FUNCTION_BLOCK FB_AxisControl
VAR_INPUT
    bControlAllowed : BOOL;// 外部控制许可
	stLimit : ST_AxisLimit;// 当前轴的限位配置
    // 仅Clamping启用：使用驱动器6061确认真实CSP/CST状态。
    bUsePhysicalModeFeedback : BOOL;
    i8ModeOfOperationDisplay : SINT;
END_VAR

VAR_IN_OUT
    AxisRef : AXIS_REF;    // TwinCAT NC轴引用
    stAxis : ST_AxisInterface;    // 单轴命令、参数和反馈接口

END_VAR

VAR
    //==========================================================
    // PLCopen功能块实例
    //==========================================================

    fbPower   : MC_Power;
    fbReset   : MC_Reset;
    fbHome    : MC_Home;
    fbStop    : MC_Stop;
    fbJog     : MC_Jog;
    fbMoveAbs : MC_MoveAbsolute;
    fbMoveRel : MC_MoveRelative;
    fbTorqueControl : MC_TorqueControl;

    // 实际转矩达到阈值后的稳定确认。
    fbTorqueReached : TON;

    //==========================================================
    // 跨Method共享的内部运行状态
    //==========================================================

    stInternal : ST_AxisControlInternal;
	//==========================================================
    // 命令上升沿
    //
    // 所有R_TRIG必须在FB主体中每周期只调用一次。
    // 各执行方法只读取Q结果，不允许再次调用R_TRIG。
    //==========================================================

    trigReset   : R_TRIG;
    trigHome    : R_TRIG;
    trigMoveAbs : R_TRIG;
    trigMoveRel : R_TRIG;
    trigJogPos  : R_TRIG;
    trigJogNeg  : R_TRIG;


END_VAR

//==============================================================
// 0. 刷新NC轴状态
//
// AXIS_REF.Status不会自动周期刷新。
// 必须在读取Status.Error、Status.ErrorId和Status.Homed之前调用。
// 每根轴、每个PLC周期只能调用一次。
//==============================================================
M_ReadAxisStatus(
    ioAxisRef := AxisRef
);

//==============================================================
// 1. 清除上一个PLC周期的瞬时结果
//
// 必须在命令检测和执行方法之前调用。
// 后续方法可以在本周期重新设置完成、终止或拒绝信号。
//==============================================================

M_ClearCycleResults(
    ioAxis := stAxis
);


//==============================================================
// 2. 更新命令上升沿
//
// 必须在M_SelectCommand和所有执行方法之前调用。
//==============================================================

M_UpdateCommandEdges(
    iCmd := stAxis.ActiveCmd
);
//==============================================================
// 3. 更新软件限位状态
//
// 必须在点动和定位执行方法之前调用。
// 相对目标、绝对目标和点动方向许可均在此处计算。
//==============================================================

M_UpdateSoftLimitState(
    iLimit    := stLimit,
    ioAxisRef := AxisRef,
    ioAxis    := stAxis
);

//==============================================================
// 4. 汇总运动状态、生成停止请求并完成命令仲裁
//==============================================================
M_UpdateCommandArbitration(
    ioAxis := stAxis
);


//==============================================================
// 5. 调用四个执行方法
//
// 虽然命令已经完成仲裁，各MC功能块仍然必须每周期调用。
//==============================================================

// MC_Power必须每周期调用；同时处理Reset
M_ExecutePowerReset(
    ioAxisRef := AxisRef,
    ioAxis    := stAxis
);

// 执行MC_Home；只响应仲裁后的HomingCmd.bHome
M_ExecuteHoming(
    ioAxisRef := AxisRef,
    ioAxis    := stAxis
);

// 执行正向和负向点动
M_ExecuteJog(
    ioAxisRef := AxisRef,
    ioAxis    := stAxis
);

// 执行绝对运动和相对运动
M_ExecutePositioning(
    ioAxisRef := AxisRef,
    ioAxis    := stAxis
);

// 执行并保持转矩控制；撤销请求时由Stop恢复位置模式
M_ExecuteTorqueControl(
    ioAxisRef := AxisRef,
    ioAxis    := stAxis
);

// Stop最后调用，保证停止具有最终优先级
M_ExecuteStop(
    ioAxisRef := AxisRef,
    ioAxis    := stAxis
);

//==============================================================
// 6. 统一更新锁存错误
//
// 必须放在四个执行方法之后，以读取本周期最新的MC输出。
// 必须放在状态更新之前，因为bReady和eMotionState需要使用
// 最新的Alarm.bError。
//==============================================================

M_UpdateError(
    ioAxisRef := AxisRef,
    ioAxis    := stAxis
);


//==============================================================
// 7. 更新基础状态
//
// 必须在M_UpdateError之后调用，确保bReady使用本周期最新错误。
// 必须在运动状态更新之前调用，保证所有基础状态先完成刷新。
//==============================================================

M_UpdateBasicState(
    ioAxisRef := AxisRef,
    ioAxis    := stAxis
);


//==============================================================
// 8. 更新唯一运动状态
//
// 必须在M_UpdateError和M_UpdateBasicState之后调用。
//==============================================================

M_UpdateMotionState(
    ioAxisRef := AxisRef,
    ioAxis    := stAxis
);

//==============================================================
// 9. 更新轴实时数据
//
// 放在本周期调用链最后，向WPF提供最新的NC轴反馈。
//==============================================================

M_UpdateAxisData(
    ioAxisRef := AxisRef,
    ioAxis    := stAxis
);
//==============================================================
// 10. 更新运动方向
//
// 使用本周期最新的：
// 1. eMotionState；
// 2. fActVelocity；
// 3. fSetVelocity。
//
// 必须放在M_UpdateMotionState和M_UpdateAxisData之后。
//==============================================================

M_UpdateMotionDirection(
    ioAxis := stAxis
);

//==============================================================
// 方法名称：M_ClearCycleResults
// 功能：清除只保持一个PLC扫描周期的结果和提示信息
//
// 注意：
// 1. 本方法必须在每个PLC周期最开始调用；
// 2. 不清除bError、nErrorID和eErrorSource等锁存报警；
// 3. 锁存报警只能在MC_Reset成功后清除。
//==============================================================

METHOD PRIVATE M_ClearCycleResults

VAR_IN_OUT
    ioAxis : ST_AxisInterface;
    // 当前轴的命令、参数和反馈接口
END_VAR
//==============================================================
// 1. 清除单周期命令结果
//==============================================================

ioAxis.State.bDone := FALSE;
ioAxis.State.bCommandAborted := FALSE;
ioAxis.State.bCmdRejected := FALSE;


//==============================================================
// 2. 清除单周期拒绝原因
//==============================================================

ioAxis.Alarm.eRejectReason :=
    E_AxisRejectReason.NoReason;


//==============================================================
// 3. 清除单周期警告
//
// 当前警告没有采用锁存方式，因此每周期重新生成。
//==============================================================

ioAxis.Alarm.bWarning := FALSE;
ioAxis.Alarm.nWarningID := 0;
END_METHOD

//==============================================================
// 执行单轴回零命令
//
// DefaultHoming使用NC轴中已经完成的参考方式、方向、速度和
// 原点传感器映射。Direct只用于仿真建立临时参考坐标；
// ForceCalibration用于绝对编码器轴，不改变当前位置。
//==============================================================
METHOD PRIVATE M_ExecuteHoming
VAR_IN_OUT
    ioAxisRef : AXIS_REF;
    ioAxis    : ST_AxisInterface;
END_VAR
VAR
    eMcHomingMode : MC_HomingMode;
    bHomeAllowed  : BOOL;
END_VAR
CASE ioAxis.ActiveSet.Homing.eCommandMode OF
    E_AxisHomeCommandMode.Direct:
        eMcHomingMode := MC_Direct;

    E_AxisHomeCommandMode.ForceCalibration:
        eMcHomingMode := MC_ForceCalibration;

    ELSE
        eMcHomingMode := MC_DefaultHoming;
END_CASE;

bHomeAllowed :=
    bControlAllowed
    AND fbPower.Status
    AND NOT ioAxis.Alarm.bError
    AND NOT stInternal.bStopExecute
    AND NOT fbStop.Busy
    AND NOT fbReset.Busy
    AND NOT fbHome.Busy
    AND NOT stInternal.bHomeExecute
    AND NOT fbJog.Busy
    AND NOT fbMoveAbs.Busy
    AND NOT fbMoveRel.Busy
    AND NOT fbTorqueControl.Busy
    AND NOT fbTorqueControl.Active
    AND NOT stInternal.bMoveAbsExecute
    AND NOT stInternal.bMoveRelExecute
    AND NOT stInternal.bTorqueExecute;

IF trigHome.Q THEN
    IF bHomeAllowed
        AND (stInternal.eRequestedCommand = E_AxisCommand.Home)
    THEN
        stInternal.bHomeExecute := TRUE;
    ELSE
        ioAxis.State.bCmdRejected := TRUE;
        ioAxis.Alarm.eRejectReason :=
            E_AxisRejectReason.HomeNotAllowed;
    END_IF;
END_IF;

IF stInternal.bStopExecute THEN
    stInternal.bHomeExecute := FALSE;
END_IF;

fbHome(
    Axis       := ioAxisRef,
    Execute    := stInternal.bHomeExecute,
    Position   := ioAxis.ActiveSet.Homing.fReferencePosition,
    HomingMode := eMcHomingMode
);

IF fbHome.Done THEN
    stInternal.bHomeExecute := FALSE;
    ioAxis.State.bDone := TRUE;

ELSIF fbHome.CommandAborted THEN
    stInternal.bHomeExecute := FALSE;
    ioAxis.State.bCommandAborted := TRUE;

ELSIF fbHome.Error THEN
    stInternal.bHomeExecute := FALSE;
END_IF;
END_METHOD

//正反点动
METHOD PRIVATE M_ExecuteJog
VAR_IN_OUT
    ioAxisRef : AXIS_REF;
    // 当前Method使用的NC轴引用

    ioAxis : ST_AxisInterface;
    // 当前Method使用的单轴接口
END_VAR

VAR
    bJogAllowed       : BOOL;
    bJogDynamicsValid : BOOL;
    bJogForward       : BOOL;
    bJogBackward      : BOOL;
    bJogCommandEdge   : BOOL;
END_VAR
//==============================================================
// 1.根据仲裁结果生成MC_Jog方向
//
// 不再直接使用两个原始按钮驱动MC_Jog，
// 防止互斥命令或高优先级命令同时进入执行层。
//==============================================================

bJogForward :=
    stInternal.eRequestedCommand = E_AxisCommand.JogPositive;

bJogBackward :=
    stInternal.eRequestedCommand = E_AxisCommand.JogNegative;
bJogCommandEdge :=
    trigJogPos.Q
    OR trigJogNeg.Q;


//==============================================================
// 2. 检查点动参数
//==============================================================

bJogDynamicsValid :=
    ioAxis.ActiveSet.Jog.fVelocity > 0.0
    AND ioAxis.ActiveSet.Jog.fAcceleration >= 0.0
    AND ioAxis.ActiveSet.Jog.fDeceleration >= 0.0;

//==============================================================
// 4. 生成点动许可
//==============================================================

bJogAllowed :=
    bControlAllowed
    AND fbPower.Status
    AND NOT ioAxis.Alarm.bError
    AND NOT stInternal.bStopExecute
    AND NOT fbStop.Busy
    AND NOT fbReset.Busy
    AND NOT fbHome.Busy
    AND NOT stInternal.bHomeExecute
    AND NOT fbMoveAbs.Busy
    AND NOT fbMoveRel.Busy
    AND NOT stInternal.bMoveAbsExecute
    AND NOT stInternal.bMoveRelExecute
    AND bJogDynamicsValid;


//==============================================================
// 5. 点动命令拒绝
//
// 只在点动按钮产生上升沿时反馈一次拒绝结果。
// 点动运行过程中进入限位区时，MC_Jog方向输入会自动撤销。
//==============================================================

IF
    bJogCommandEdge
    AND ioAxis.ActiveCmd.bJogPos
    AND ioAxis.ActiveCmd.bJogNeg
THEN

    ioAxis.State.bCmdRejected := TRUE;

    ioAxis.Alarm.eRejectReason :=
        E_AxisRejectReason.JogDirectionConflict;


ELSIF
    bJogCommandEdge
    AND NOT bJogDynamicsValid
THEN

    ioAxis.State.bCmdRejected := TRUE;

    ioAxis.Alarm.eRejectReason :=
        E_AxisRejectReason.InvalidDynamics;


ELSIF
    bJogCommandEdge
    AND stInternal.stSoftLimitResult.bEnabled
    AND NOT stInternal.stSoftLimitResult.bConfigValid
THEN

    ioAxis.State.bCmdRejected := TRUE;

    ioAxis.Alarm.eRejectReason :=
        E_AxisRejectReason.SoftLimitConfigInvalid;


ELSIF
    bJogCommandEdge
    AND stInternal.stSoftLimitResult.bEnabled
    AND NOT stInternal.stSoftLimitResult.bReferenceValid
THEN

    ioAxis.State.bCmdRejected := TRUE;

    ioAxis.Alarm.eRejectReason :=
        E_AxisRejectReason.NotHomed;


ELSIF
    bJogCommandEdge
    AND
    (
        (
            ioAxis.ActiveCmd.bJogPos
            AND NOT stInternal.stSoftLimitResult.bJogPositiveAllowed
        )
        OR
        (
            ioAxis.ActiveCmd.bJogNeg
            AND NOT stInternal.stSoftLimitResult.bJogNegativeAllowed
        )
    )
THEN

    ioAxis.State.bCmdRejected := TRUE;

    ioAxis.Alarm.eRejectReason :=
        E_AxisRejectReason.TargetOutOfLimit;


ELSIF
    bJogCommandEdge
    AND NOT bJogAllowed
THEN

    ioAxis.State.bCmdRejected := TRUE;

    ioAxis.Alarm.eRejectReason :=
        E_AxisRejectReason.AxisNotReady;

END_IF;


//==============================================================
// 6. 周期调用MC_Jog
//==============================================================

fbJog(
    Axis := ioAxisRef,

    // 正向点动同时受到通用许可和正向软限位许可约束
    JogForward :=
        bJogAllowed
        AND bJogForward
        AND stInternal.stSoftLimitResult.bJogPositiveAllowed,

    // 负向点动同时受到通用许可和负向软限位许可约束
    JogBackwards :=
        bJogAllowed
        AND bJogBackward
        AND stInternal.stSoftLimitResult.bJogNegativeAllowed,

    Mode         := MC_JOGMODE_CONTINOUS,
    Position     := 0.0,
    Velocity     := ioAxis.ActiveSet.Jog.fVelocity,
    Acceleration := ioAxis.ActiveSet.Jog.fAcceleration,
    Deceleration := ioAxis.ActiveSet.Jog.fDeceleration,
    Jerk         := 0.0
);


//==============================================================
// 7. 点动被其他命令打断
//==============================================================

IF fbJog.CommandAborted THEN
    ioAxis.State.bCommandAborted := TRUE;
END_IF;
END_METHOD

//相对、绝对定位运动
METHOD PRIVATE M_ExecutePositioning
VAR_IN_OUT
    ioAxisRef : AXIS_REF;
    ioAxis    : ST_AxisInterface;
END_VAR

VAR
    bPositionAllowed       : BOOL;
    bPositionDynamicsValid : BOOL;
END_VAR
//==============================================================
// 1. 绝对/相对运动命令上升沿
//==============================================================



//==============================================================
// 2. 定位参数检查
//==============================================================

bPositionDynamicsValid :=
    ioAxis.ActiveSet.Position.fVelocity > 0.0
    AND ioAxis.ActiveSet.Position.fAcceleration >= 0.0
    AND ioAxis.ActiveSet.Position.fDeceleration >= 0.0;


//==============================================================
// 3. 统一定位许可
//==============================================================

bPositionAllowed :=
    bControlAllowed
    AND fbPower.Status
    AND ioAxis.State.bPositionModeReady
    AND NOT ioAxis.Alarm.bError
    AND NOT stInternal.bStopExecute
    AND NOT fbStop.Busy
    AND NOT fbReset.Busy
    AND NOT fbHome.Busy
    AND NOT stInternal.bHomeExecute
    AND NOT fbJog.Busy
    AND NOT ioAxis.ActiveCmd.bJogPos
    AND NOT ioAxis.ActiveCmd.bJogNeg
    AND NOT fbMoveAbs.Busy
    AND NOT fbMoveRel.Busy
    AND NOT stInternal.bMoveAbsExecute
    AND NOT stInternal.bMoveRelExecute;


//==============================================================
// 4. 接受或拒绝定位命令
//==============================================================

IF trigMoveAbs.Q AND trigMoveRel.Q THEN

    // 绝对和相对命令同时触发
    ioAxis.State.bCmdRejected := TRUE;

    ioAxis.Alarm.eRejectReason :=
        E_AxisRejectReason.CommandConflict;


ELSIF trigMoveAbs.Q OR trigMoveRel.Q THEN

    //==========================================================
    // 4.1 轴当前不允许定位
    //==========================================================

    IF NOT bPositionAllowed THEN

        ioAxis.State.bCmdRejected := TRUE;

        ioAxis.Alarm.eRejectReason :=
            E_AxisRejectReason.AxisNotReady;


    //==========================================================
    // 4.2 动态参数错误
    //==========================================================

    ELSIF NOT bPositionDynamicsValid THEN

        ioAxis.State.bCmdRejected := TRUE;

        ioAxis.Alarm.eRejectReason :=
            E_AxisRejectReason.InvalidDynamics;


    //==========================================================
    // 4.3 软件限位配置错误
    //==========================================================

    ELSIF
        stInternal.stSoftLimitResult.bEnabled
        AND NOT stInternal.stSoftLimitResult.bConfigValid
    THEN

        ioAxis.State.bCmdRejected := TRUE;

        ioAxis.Alarm.eRejectReason :=
            E_AxisRejectReason.SoftLimitConfigInvalid;


    //==========================================================
    // 4.4 尚未建立有效坐标基准
    //==========================================================

    ELSIF
        stInternal.stSoftLimitResult.bEnabled
        AND NOT stInternal.stSoftLimitResult.bReferenceValid
    THEN

        ioAxis.State.bCmdRejected := TRUE;

        ioAxis.Alarm.eRejectReason :=
            E_AxisRejectReason.NotHomed;


    //==========================================================
    // 4.5 绝对目标超出软件限位
    //==========================================================

    ELSIF
        stInternal.eRequestedCommand = E_AxisCommand.MoveAbsolute
        AND NOT stInternal.stSoftLimitResult.bAbsoluteTargetValid
    THEN

        ioAxis.State.bCmdRejected := TRUE;

        ioAxis.Alarm.eRejectReason :=
            E_AxisRejectReason.TargetOutOfLimit;


    //==========================================================
    // 4.6 相对运动最终目标超出软件限位
    //==========================================================

    ELSIF
        stInternal.eRequestedCommand = E_AxisCommand.MoveRelative
        AND NOT stInternal.stSoftLimitResult.bRelativeTargetValid
    THEN

        ioAxis.State.bCmdRejected := TRUE;

        ioAxis.Alarm.eRejectReason :=
            E_AxisRejectReason.TargetOutOfLimit;


    //==========================================================
    // 4.7 接受绝对运动
    //==========================================================

    ELSIF
        stInternal.eRequestedCommand = E_AxisCommand.MoveAbsolute
    THEN

        stInternal.bMoveAbsExecute := TRUE;


    //==========================================================
    // 4.8 接受相对运动
    //==========================================================

    ELSIF
        stInternal.eRequestedCommand = E_AxisCommand.MoveRelative
    THEN

        stInternal.bMoveRelExecute := TRUE;


    //==========================================================
    // 4.9 请求被高优先级命令覆盖
    //==========================================================

    ELSE

        ioAxis.State.bCmdRejected := TRUE;

        ioAxis.Alarm.eRejectReason :=
            E_AxisRejectReason.AxisNotReady;

    END_IF;

END_IF;


//==============================================================
// 5. Stop开始后撤销普通运动Execute
//==============================================================

IF stInternal.bStopExecute THEN
    stInternal.bHomeExecute := FALSE;
    stInternal.bMoveAbsExecute := FALSE;
    stInternal.bMoveRelExecute := FALSE;
    stInternal.bTorqueExecute := FALSE;
END_IF;


//==============================================================
// 6. 周期调用MC_MoveAbsolute
//==============================================================

fbMoveAbs(
    Axis         := ioAxisRef,
    Execute      := stInternal.bMoveAbsExecute,
    Position     := ioAxis.ActiveSet.Position.fAbsolutePosition,
    Velocity     := ioAxis.ActiveSet.Position.fVelocity,
    Acceleration := ioAxis.ActiveSet.Position.fAcceleration,
    Deceleration := ioAxis.ActiveSet.Position.fDeceleration,
    Jerk         := 0.0,
    BufferMode   := MC_Aborting
);


//==============================================================
// 7. 周期调用MC_MoveRelative
//==============================================================

fbMoveRel(
    Axis         := ioAxisRef,
    Execute      := stInternal.bMoveRelExecute,
    Distance     := ioAxis.ActiveSet.Position.fRelativeDistance,
    Velocity     := ioAxis.ActiveSet.Position.fVelocity,
    Acceleration := ioAxis.ActiveSet.Position.fAcceleration,
    Deceleration := ioAxis.ActiveSet.Position.fDeceleration,
    Jerk         := 0.0,
    BufferMode   := MC_Aborting
);


//==============================================================
// 8. 绝对运动结果
//==============================================================

IF fbMoveAbs.Done THEN

    stInternal.bMoveAbsExecute := FALSE;
    ioAxis.State.bDone := TRUE;

ELSIF fbMoveAbs.CommandAborted THEN

    stInternal.bMoveAbsExecute := FALSE;
    ioAxis.State.bCommandAborted := TRUE;

ELSIF fbMoveAbs.Error THEN

    stInternal.bMoveAbsExecute := FALSE;

END_IF;


//==============================================================
// 9. 相对运动结果
//==============================================================

IF fbMoveRel.Done THEN

    stInternal.bMoveRelExecute := FALSE;
    ioAxis.State.bDone := TRUE;

ELSIF fbMoveRel.CommandAborted THEN

    stInternal.bMoveRelExecute := FALSE;
    ioAxis.State.bCommandAborted := TRUE;

ELSIF fbMoveRel.Error THEN

    stInternal.bMoveRelExecute := FALSE;

END_IF;
END_METHOD

//==============================================================
// 执行持续型转矩控制。
// 撤销bTorqueControl后，命令仲裁会请求MC_Stop，
// 由NC将轴从CST恢复到位置相关模式。
//==============================================================
METHOD PRIVATE M_ExecuteTorqueControl
VAR_IN_OUT
    ioAxisRef : AXIS_REF;
    ioAxis    : ST_AxisInterface;
END_VAR

VAR
    bTorqueParametersValid : BOOL;
    bTorqueAllowed         : BOOL;
END_VAR
//==============================================================
// 1. 参数和执行许可
//==============================================================
bTorqueParametersValid :=
    ioAxis.ActiveSet.Torque.fMaxAbsTorquePercent > 0.0
    AND ABS(ioAxis.ActiveSet.Torque.fTargetTorquePercent)
        <= ioAxis.ActiveSet.Torque.fMaxAbsTorquePercent
    AND ioAxis.ActiveSet.Torque.fTorqueRampPercentPerSecond > 0.0
    AND ioAxis.ActiveSet.Torque.fVelocityLimitHigh > 0.0
    AND ioAxis.ActiveSet.Torque.fVelocityLimitLow < 0.0
    AND ioAxis.ActiveSet.Torque.fVelocityLimitHigh
        > ioAxis.ActiveSet.Torque.fVelocityLimitLow;

bTorqueAllowed :=
    bControlAllowed
    AND fbPower.Status
    AND NOT ioAxis.Alarm.bError
    AND NOT stInternal.bStopExecute
    AND NOT fbStop.Busy
    AND NOT fbReset.Busy
    AND NOT fbHome.Busy
    AND NOT stInternal.bHomeExecute
    AND NOT fbJog.Busy
    AND NOT fbMoveAbs.Busy
    AND NOT fbMoveRel.Busy
    AND NOT stInternal.bMoveAbsExecute
    AND NOT stInternal.bMoveRelExecute;

//==============================================================
// 2. 接受、保持或撤销转矩命令
//==============================================================
IF
    NOT ioAxis.ActiveCmd.bTorqueControl
    OR
    (stInternal.eRequestedCommand <> E_AxisCommand.TorqueControl)
THEN
    stInternal.bTorqueExecute := FALSE;

ELSIF NOT stInternal.bTorqueExecute THEN
    IF NOT bTorqueAllowed THEN
        ioAxis.State.bCmdRejected := TRUE;
        ioAxis.Alarm.eRejectReason :=
            E_AxisRejectReason.AxisNotReady;

    ELSIF NOT bTorqueParametersValid THEN
        ioAxis.State.bCmdRejected := TRUE;
        ioAxis.Alarm.eRejectReason :=
            E_AxisRejectReason.InvalidDynamics;

    ELSE
        stInternal.bTorqueExecute := TRUE;
    END_IF;
END_IF;

//==============================================================
// 3. 周期调用MC_TorqueControl
//==============================================================
fbTorqueControl(
    Axis              := ioAxisRef,
    Execute           := stInternal.bTorqueExecute,
    ContinuousUpdate  := TRUE,
    Relative          := FALSE,
    Torque            := ioAxis.ActiveSet.Torque.fTargetTorquePercent,
    TorqueRamp        := ioAxis.ActiveSet.Torque.fTorqueRampPercentPerSecond,
    VelocityLimitHigh := ioAxis.ActiveSet.Torque.fVelocityLimitHigh,
    VelocityLimitLow  := ioAxis.ActiveSet.Torque.fVelocityLimitLow,
    BufferMode        := MC_Aborting
);

//==============================================================
// 4. 实际转矩稳定确认
//==============================================================
fbTorqueReached(
    IN :=
        fbTorqueControl.Active
        AND
        (
            ABS(ioAxis.Data.fActTorque)
            >= ioAxis.ActiveSet.Torque.fReachedMinAbsTorquePercent
        ),
    PT := ioAxis.ActiveSet.Torque.tReachedStableTime
);

ioAxis.State.bTorqueReached := fbTorqueReached.Q;
ioAxis.State.bTorqueControlActive := fbTorqueControl.Active;

//==============================================================
// 5. 发布当前控制模式
//==============================================================
IF bUsePhysicalModeFeedback THEN
    // Clamping必须以驱动器6061为准，不能由PLCopen FB内部状态推断。
    CASE i8ModeOfOperationDisplay OF
        8:
            ioAxis.State.eControlMode := E_AxisControlMode.Position;
        10:
            ioAxis.State.eControlMode := E_AxisControlMode.Torque;
        ELSE
            ioAxis.State.eControlMode := E_AxisControlMode.Undefined;
    END_CASE;
ELSE
    IF fbTorqueControl.Active OR fbTorqueControl.Busy THEN
        ioAxis.State.eControlMode := E_AxisControlMode.Torque;
    ELSIF
        fbPower.Status
        AND NOT stInternal.bStopExecute
        AND NOT fbStop.Busy
    THEN
        ioAxis.State.eControlMode := E_AxisControlMode.Position;
    ELSE
        ioAxis.State.eControlMode := E_AxisControlMode.Undefined;
    END_IF;
END_IF;

ioAxis.State.bPositionModeReady :=
    fbPower.Status
    AND (ioAxis.State.eControlMode = E_AxisControlMode.Position)
    AND NOT stInternal.bStopExecute
    AND NOT fbStop.Busy;

ioAxis.State.bTorqueModeReady :=
    fbTorqueControl.Active
    AND (ioAxis.State.eControlMode = E_AxisControlMode.Torque);

//==============================================================
// 6. 功能块结果
//==============================================================
IF fbTorqueControl.CommandAborted THEN
    stInternal.bTorqueExecute := FALSE;
    ioAxis.State.bCommandAborted := TRUE;
ELSIF fbTorqueControl.Error THEN
    stInternal.bTorqueExecute := FALSE;
END_IF;
END_METHOD

//调用 MC_Power和MC_Reset
METHOD PRIVATE M_ExecutePowerReset
VAR_IN_OUT
    ioAxisRef : AXIS_REF;
    ioAxis    : ST_AxisInterface;
END_VAR

VAR
    bPowerEnable  : BOOL; // 实际送入MC_Power的Enable
    bResetAllowed : BOOL; // 当前是否允许复位	
END_VAR
//==============================================================
// 1. 生成MC_Power实际使能信号
//
// 外部要求使能时正常保持使能。
// 运动中撤销使能时，先保持使能完成MC_Stop。
//==============================================================

bPowerEnable :=
    ioAxis.ActiveCmd.bEnable
    OR
    (
        (stInternal.bStopExecute OR fbStop.Busy)
        AND fbPower.Status
    );


//==============================================================
// 2. 周期调用MC_Power
//==============================================================

fbPower(
    Axis            := ioAxisRef,
    Enable          := bPowerEnable,
    Enable_Positive := TRUE,
    Enable_Negative := TRUE,
    Override        := 100.0
);



//==============================================================
// 3. Reset许可
//
// 运动、点动和停止过程中不允许Reset。
//==============================================================

bResetAllowed :=
    NOT stInternal.bMotionActive
    AND NOT stInternal.bStopExecute
    AND NOT fbStop.Busy;

//==============================================================
// 4. 周期调用MC_Reset
//
// Reset必须同时满足：
// 1. 已被M_SelectCommand选中；
// 2. 当前轴状态允许复位。
//==============================================================

fbReset(
    Axis := ioAxisRef,
    Execute :=
        (stInternal.eRequestedCommand = E_AxisCommand.Reset)
        AND bResetAllowed
);


//==============================================================
// 5. Reset命令被拒绝
//==============================================================

IF
    (stInternal.eRequestedCommand = E_AxisCommand.Reset)
    AND NOT bResetAllowed
THEN
    ioAxis.State.bCmdRejected := TRUE;

    ioAxis.Alarm.eRejectReason :=
        E_AxisRejectReason.ResetDuringMotion;
END_IF;

//==============================================================
// 6. Reset成功
//
// 清除PLC锁存的轴报警。
//==============================================================

IF fbReset.Done THEN

    ioAxis.Alarm.bError       := FALSE;
    ioAxis.Alarm.nErrorID     := 0;
    ioAxis.Alarm.eErrorSource :=
        E_AxisErrorSource.NoError;

    ioAxis.State.bDone := TRUE;

END_IF;
END_METHOD

//处理最高优先级停止和 MC_Stop
METHOD PRIVATE M_ExecuteStop
VAR_IN_OUT
    ioAxisRef : AXIS_REF;
    ioAxis    : ST_AxisInterface;
END_VAR

VAR
    fStopDeceleration : LREAL;//停止声明
END_VAR
//==============================================================
// 1. Stop开始后撤销定位和转矩Execute
//==============================================================
IF stInternal.bStopExecute THEN
    stInternal.bHomeExecute := FALSE;
    stInternal.bMoveAbsExecute := FALSE;
    stInternal.bMoveRelExecute := FALSE;
    stInternal.bTorqueExecute := FALSE;
END_IF;


//==============================================================
// 2. 选择停止减速度
//
// 当前沿用位置运动减速度。
// 如果配置值小于0，则使用0，让NC采用默认减速度。
//==============================================================
fStopDeceleration :=
    ioAxis.ActiveSet.Position.fDeceleration;

IF fStopDeceleration < 0.0 THEN
    fStopDeceleration := 0.0;
END_IF;


//==============================================================
// 3. 每周期调用MC_Stop
//==============================================================
fbStop(
    Axis         := ioAxisRef,
    Execute      := stInternal.bStopExecute,
    Deceleration := fStopDeceleration,
    Jerk         := 0.0
);


//==============================================================
// 4. 发布MC_Stop专用状态
//
// 不使用通用State.bDone，避免与MoveAbs、MoveRel等完成信号混淆。
//==============================================================
ioAxis.State.bStopDone :=
    fbStop.Done;

// Done仅代表停住；释放Execute并等待Busy结束后才能掉使能。
ioAxis.State.bStopReleased :=
    NOT stInternal.bStopExecute
    AND NOT fbStop.Busy;

ioAxis.State.bStopError :=
    fbStop.Error;

ioAxis.State.nStopErrorID :=
    fbStop.ErrorID;


//==============================================================
// 5. 外部停止请求释放后，解除MC_Stop锁定
//==============================================================
IF
    fbStop.Done
    AND NOT stInternal.bStopRequest
THEN
    stInternal.bStopExecute := FALSE;
END_IF;


//==============================================================
// 6. Stop错误
//
// 即使停止发生错误，也要撤销内部Execute，
// 错误信息由State和Alarm继续对外发布。
//==============================================================
IF fbStop.Error THEN
    stInternal.bStopExecute := FALSE;
END_IF;
END_METHOD

// 刷新NC轴状态。每根轴、每周期只调用一次。
METHOD PRIVATE M_ReadAxisStatus
VAR_IN_OUT
    ioAxisRef : AXIS_REF;
END_VAR
ioAxisRef.ReadStatus();
END_METHOD

//==============================================================
// 方法名称：M_SelectCommand
// 功能：
// 1. 识别外部BOOL命令；
// 2. 将多个BOOL命令转换成唯一E_AxisCommand；
// 3. 实现停止、复位、点动、定位之间的优先级；
// 4. 发现互斥命令时返回NoCommand。
//
// 本方法只进行命令选择，不调用任何MC功能块。
//==============================================================

METHOD PRIVATE M_SelectCommand : E_AxisCommand

VAR_INPUT
    bStopRequest  : BOOL; // 停止请求，最高优先级
    bResetPulse   : BOOL; // 复位命令上升沿

    bHomePulse    : BOOL; // 回零命令上升沿

    bTorqueControl : BOOL; // 持续型转矩控制请求

    bJogPositive  : BOOL; // 正向点动保持信号
    bJogNegative  : BOOL; // 负向点动保持信号

    bMoveAbsPulse : BOOL; // 绝对运动命令上升沿
    bMoveRelPulse : BOOL; // 相对运动命令上升沿
END_VAR
// 默认本周期没有有效命令
M_SelectCommand := E_AxisCommand.NoCommand;


//==============================================================
// 1. 停止命令
//
// Stop具有最高优先级，可以覆盖复位、点动和定位命令。
// bStopRequest还包括撤销控制许可和运动中撤销使能。
//==============================================================

IF bStopRequest THEN

    M_SelectCommand := E_AxisCommand.Stop;


//==============================================================
// 2. 复位命令
//
// Reset使用上升沿，只在触发周期返回Reset。
// 是否允许复位仍由M_ExecutePowerReset检查。
//==============================================================

ELSIF bResetPulse THEN

    M_SelectCommand := E_AxisCommand.Reset;


//==============================================================
// 3. 回零命令
//==============================================================

ELSIF bHomePulse THEN

    M_SelectCommand := E_AxisCommand.Home;


//==============================================================
// 4. 转矩控制
//==============================================================

ELSIF bTorqueControl THEN

    M_SelectCommand := E_AxisCommand.TorqueControl;


//==============================================================
// 4. 点动方向冲突
//
// 正向点动和负向点动同时成立时不选择任何方向。
// 具体拒绝原因由M_ExecuteJog写入状态和报警接口。
//==============================================================

ELSIF bJogPositive AND bJogNegative THEN

    M_SelectCommand := E_AxisCommand.NoCommand;


//==============================================================
// 5. 正向和负向点动
//
// 点动是保持型命令：
// 按钮保持TRUE时，每周期持续返回对应点动命令；
// 松开按钮后返回NoCommand，MC_Jog开始减速停止。
//==============================================================

ELSIF bJogPositive THEN

    M_SelectCommand := E_AxisCommand.JogPositive;

ELSIF bJogNegative THEN

    M_SelectCommand := E_AxisCommand.JogNegative;


//==============================================================
// 6. 定位命令冲突
//
// 绝对运动和相对运动在同一扫描周期同时触发时，
// 不选择任何定位命令。
// 具体拒绝原因由M_ExecutePositioning写入反馈。
//==============================================================

ELSIF bMoveAbsPulse AND bMoveRelPulse THEN

    M_SelectCommand := E_AxisCommand.NoCommand;


//==============================================================
// 7. 绝对运动和相对运动
//==============================================================

ELSIF bMoveAbsPulse THEN

    M_SelectCommand := E_AxisCommand.MoveAbsolute;

ELSIF bMoveRelPulse THEN

    M_SelectCommand := E_AxisCommand.MoveRelative;

END_IF;
END_METHOD

//==============================================================
// 方法名称：M_UpdateAxisData
// 功能：
// 1. 从AXIS_REF.NcToPlc读取NC轴实时数据；
// 2. 写入ST_AxisData，供PLC程序和WPF读取；
// 3. 集中处理后续可能增加的单位换算。
//
// 调用位置：
// 放在所有命令执行、错误和状态更新之后，每周期调用一次。
//==============================================================

METHOD PRIVATE M_UpdateAxisData

VAR_IN_OUT
    ioAxisRef : AXIS_REF;
    // 当前TwinCAT NC轴引用

    ioAxis : ST_AxisInterface;
    // 当前单轴数据反馈接口
END_VAR
//==============================================================
// 1. 位置数据
//==============================================================

// NC轴设定位置
ioAxis.Data.fSetPosition :=
    ioAxisRef.NcToPlc.SetPos;

// 编码器反馈的实际位置
ioAxis.Data.fActPosition :=
    ioAxisRef.NcToPlc.ActPos;

// 当前运动的目标位置
ioAxis.Data.fTargetPosition :=
    ioAxisRef.NcToPlc.TargetPos;


//==============================================================
// 2. 速度数据
//==============================================================

// NC轴设定速度
ioAxis.Data.fSetVelocity :=
    ioAxisRef.NcToPlc.SetVelo;

// 编码器反馈的实际速度
ioAxis.Data.fActVelocity :=
    ioAxisRef.NcToPlc.ActVelo;


//==============================================================
// 3. 加速度数据
//==============================================================

// NC轴设定加速度
ioAxis.Data.fSetAcceleration :=
    ioAxisRef.NcToPlc.SetAcc;

// NC轴实际加速度
ioAxis.Data.fActAcceleration :=
    ioAxisRef.NcToPlc.ActAcc;


//==============================================================
// 4. 跟随误差
//
// 带方向的位置偏差。
//==============================================================

ioAxis.Data.fFollowingError :=
    ioAxisRef.NcToPlc.PosDiff;


//==============================================================
// 5. 转矩数据
//
// 是否为实际物理转矩、百分比或归一化值，
// 取决于驱动器和NC轴的配置。
//==============================================================

ioAxis.Data.fSetTorque :=
    ioAxisRef.NcToPlc.SetTorque;

ioAxis.Data.fActTorque :=
    ioAxisRef.NcToPlc.ActTorque;


//==============================================================
// 6. 电机转速
//
// 当前缺少“每转对应多少工程单位”的换算参数，
// 因此暂不计算实际rpm。
//==============================================================

ioAxis.Data.fActRpm := 0.0;
END_METHOD

//==============================================================
// 方法名称：M_UpdateBasicState
// 功能：
// 1. 汇总各PLCopen功能块的Busy状态；
// 2. 更新轴使能、忙碌、活动、准备完成和回零状态；
// 3. 为WPF提供统一的基础状态反馈。
//
// 调用位置：
// 必须放在四个执行方法和M_UpdateError之后。
//==============================================================

METHOD PRIVATE M_UpdateBasicState

VAR_IN_OUT
    ioAxisRef : AXIS_REF;
    // 当前TwinCAT NC轴引用

    ioAxis : ST_AxisInterface;
    // 当前单轴状态和报警接口
END_VAR
//==============================================================
// 1. 汇总轴忙碌状态
//
// 除PLCopen功能块的Busy外，还包含三个Execute锁存信号，
// 避免命令已经接受但Busy尚未建立时出现一周期状态空缺。
//==============================================================

stInternal.bAnyBusy :=
    fbReset.Busy
    OR fbHome.Busy
    OR stInternal.bHomeExecute
    OR fbStop.Busy
    OR stInternal.bStopExecute
    OR fbJog.Busy
    OR fbMoveAbs.Busy
    OR fbMoveRel.Busy
    OR fbTorqueControl.Busy
    OR stInternal.bMoveAbsExecute
    OR stInternal.bMoveRelExecute
    OR stInternal.bTorqueExecute;


//==============================================================
// 2. 更新实际使能状态
//
// 采用MC_Power.Status，而不是外部bEnable请求。
//==============================================================

ioAxis.State.bPowerStatus :=
    fbPower.Status;


//==============================================================
// 3. 更新忙碌状态
//
// 复位、停止、点动或定位过程中均视为Busy。
//==============================================================

ioAxis.State.bBusy :=
    stInternal.bAnyBusy;


//==============================================================
// 4. 更新有效运动状态
//
// bActive表示NC轴当前存在实际运动或停止过程。
// 不包含仅已锁存、但PLCopen Busy尚未建立的命令。
//==============================================================

ioAxis.State.bActive :=
    fbJog.Busy
    OR fbHome.Busy
    OR fbMoveAbs.Busy
    OR fbMoveRel.Busy
    OR fbTorqueControl.Active
    OR fbStop.Busy;


//==============================================================
// 5. 更新轴准备状态
//
// 满足以下全部条件才允许接受新的普通运动命令：
// 1. 轴已经实际使能；
// 2. 外部控制许可有效；
// 3. 没有锁存错误；
// 4. 当前没有正在执行的命令。
//==============================================================

ioAxis.State.bReady :=
    fbPower.Status
    AND bControlAllowed
    AND NOT ioAxis.Alarm.bError
    AND NOT stInternal.bAnyBusy;


//==============================================================
// 6. 更新回零状态
//
// MC_Home和NC轴状态共同维护该标志。
//==============================================================

ioAxis.State.bHomed :=
    ioAxisRef.Status.Homed;
END_METHOD

//==============================================================
// 汇总运动状态、生成停止请求、选择唯一命令并锁存停止。
//==============================================================
METHOD PRIVATE M_UpdateCommandArbitration
VAR_IN_OUT
    ioAxis : ST_AxisInterface;
END_VAR
// Execute已锁存但Busy尚未建立时，同样视为运动有效。
stInternal.bMotionActive :=
    fbJog.Busy
    OR fbHome.Busy
    OR fbMoveAbs.Busy
    OR fbMoveRel.Busy
    OR fbTorqueControl.Active
    OR fbTorqueControl.Busy
    OR stInternal.bMoveAbsExecute
    OR stInternal.bMoveRelExecute
    OR stInternal.bHomeExecute
    OR stInternal.bTorqueExecute;


// 外部Stop、运动中撤销控制许可或撤销使能均请求停止。
stInternal.bStopRequest :=
    ioAxis.ActiveCmd.bStop
    OR
    (
        (fbTorqueControl.Active OR fbTorqueControl.Busy)
        AND NOT ioAxis.ActiveCmd.bTorqueControl
    )
    OR
    (
        NOT bControlAllowed
        AND stInternal.bMotionActive
    )
    OR
    (
        NOT ioAxis.ActiveCmd.bEnable
        AND stInternal.bMotionActive
    );


// 优先级：Stop > Reset > Torque > Jog > MoveAbsolute/MoveRelative。
stInternal.eRequestedCommand := M_SelectCommand(
    bStopRequest := stInternal.bStopRequest,
    bResetPulse := trigReset.Q,
    bHomePulse := trigHome.Q,
    bTorqueControl := ioAxis.ActiveCmd.bTorqueControl,
    bJogPositive := ioAxis.ActiveCmd.bJogPos,
    bJogNegative := ioAxis.ActiveCmd.bJogNeg,
    bMoveAbsPulse := trigMoveAbs.Q,
    bMoveRelPulse := trigMoveRel.Q
);


// Stop一旦被选中，保持Execute直至停止完成并释放外部Stop。
IF
    (stInternal.eRequestedCommand = E_AxisCommand.Stop)
    AND fbPower.Status
THEN
    stInternal.bStopExecute := TRUE;
END_IF;
END_METHOD

//==============================================================
// 方法名称：M_UpdateCommandEdges
// 功能：统一更新单轴命令的上升沿检测结果
//
// 注意：
// 1. 每个R_TRIG实例每周期只能在本方法中调用一次；
// 2. Reset、绝对运动、相对运动使用上升沿触发；
// 3. 点动使用持续信号，上升沿仅用于判断命令是否被拒绝；
// 4. Enable和Stop是持续型信号，不需要R_TRIG。
//==============================================================

METHOD PRIVATE M_UpdateCommandEdges

VAR_INPUT
    iCmd : ST_AxisCmd;
    // 当前轴的原始命令
    // 结构体较小，使用VAR_INPUT传递不会造成明显开销
END_VAR
//==============================================================
// 1. 错误复位命令上升沿
//==============================================================

trigReset(
    CLK := iCmd.bReset
);


//==============================================================
// 2. 回零命令上升沿
//==============================================================

trigHome(
    CLK := iCmd.bHome
);


//==============================================================
// 3. 绝对运动命令上升沿
//==============================================================

trigMoveAbs(
    CLK := iCmd.bMoveAbs
);


//==============================================================
// 3. 相对运动命令上升沿
//==============================================================

trigMoveRel(
    CLK := iCmd.bMoveRel
);


//==============================================================
// 4. 正向点动按钮上升沿
//
// MC_Jog仍然使用bJogPos持续电平；
// 本上升沿只用于产生命令拒绝反馈。
//==============================================================

trigJogPos(
    CLK := iCmd.bJogPos
);


//==============================================================
// 5. 负向点动按钮上升沿
//==============================================================

trigJogNeg(
    CLK := iCmd.bJogNeg
);
END_METHOD

//==============================================================
// 方法名称：M_UpdateError
// 功能：
// 1. 汇总NC轴和各PLCopen功能块错误；
// 2. 根据优先级选择当前显示的错误；
// 3. 将错误锁存到单轴报警接口。
//
// 错误优先级：
// NC轴 > Stop > Power > Reset > Jog > 绝对运动 > 相对运动
//
// 注意：
// 1. 本方法不主动清除错误；
// 2. 错误只能在MC_Reset成功后清除；
// 3. 没有新错误时保持原报警不变。
//==============================================================

METHOD PRIVATE M_UpdateError

VAR_IN_OUT
    ioAxisRef : AXIS_REF;
    // 当前TwinCAT NC轴引用

    ioAxis : ST_AxisInterface;
    // 当前轴的状态和报警接口
END_VAR
//==============================================================
// 1. NC轴错误
//
// NC轴本体错误优先级最高。
//==============================================================

IF ioAxisRef.Status.Error THEN

    ioAxis.Alarm.bError := TRUE;
    ioAxis.Alarm.nErrorID :=
        ioAxisRef.Status.ErrorId;

    ioAxis.Alarm.eErrorSource :=
        E_AxisErrorSource.NcAxis;


//==============================================================
// 2. MC_Stop错误
//==============================================================

ELSIF fbStop.Error THEN

    ioAxis.Alarm.bError := TRUE;
    ioAxis.Alarm.nErrorID :=
        fbStop.ErrorID;

    ioAxis.Alarm.eErrorSource :=
        E_AxisErrorSource.Stop;


//==============================================================
// 3. MC_Power错误
//==============================================================

ELSIF fbPower.Error THEN

    ioAxis.Alarm.bError := TRUE;
    ioAxis.Alarm.nErrorID :=
        fbPower.ErrorID;

    ioAxis.Alarm.eErrorSource :=
        E_AxisErrorSource.Power;


//==============================================================
// 4. MC_Reset错误
//==============================================================

ELSIF fbReset.Error THEN

    ioAxis.Alarm.bError := TRUE;
    ioAxis.Alarm.nErrorID :=
        fbReset.ErrorID;

    ioAxis.Alarm.eErrorSource :=
        E_AxisErrorSource.Reset;


//==============================================================
// 5. MC_Home错误
//==============================================================

ELSIF fbHome.Error THEN

    ioAxis.Alarm.bError := TRUE;
    ioAxis.Alarm.nErrorID :=
        fbHome.ErrorID;

    ioAxis.Alarm.eErrorSource :=
        E_AxisErrorSource.Home;


//==============================================================
// 6. MC_TorqueControl错误
//==============================================================

ELSIF fbTorqueControl.Error THEN

    ioAxis.Alarm.bError := TRUE;
    ioAxis.Alarm.nErrorID :=
        fbTorqueControl.ErrorID;

    ioAxis.Alarm.eErrorSource :=
        E_AxisErrorSource.TorqueControl;


//==============================================================
// 6. MC_Jog错误
//==============================================================

ELSIF fbJog.Error THEN

    ioAxis.Alarm.bError := TRUE;
    ioAxis.Alarm.nErrorID :=
        fbJog.ErrorID;

    ioAxis.Alarm.eErrorSource :=
        E_AxisErrorSource.Jog;


//==============================================================
// 7. MC_MoveAbsolute错误
//==============================================================

ELSIF fbMoveAbs.Error THEN

    ioAxis.Alarm.bError := TRUE;
    ioAxis.Alarm.nErrorID :=
        fbMoveAbs.ErrorID;

    ioAxis.Alarm.eErrorSource :=
        E_AxisErrorSource.MoveAbsolute;


//==============================================================
// 8. MC_MoveRelative错误
//==============================================================

ELSIF fbMoveRel.Error THEN

    ioAxis.Alarm.bError := TRUE;
    ioAxis.Alarm.nErrorID :=
        fbMoveRel.ErrorID;

    ioAxis.Alarm.eErrorSource :=
        E_AxisErrorSource.MoveRelative;

END_IF;
END_METHOD

//==============================================================
// 方法名称：M_UpdateMotionDirection
//
// 功能：
// 1. 根据轴当前运动状态判断是否需要输出运动方向；
// 2. 优先使用NC实际速度判断方向；
// 3. 运动刚启动、实际速度尚未建立时，使用NC设定速度辅助判断；
// 4. 停止、故障、未使能等状态统一输出None；
// 5. 不使用目标位置，避免中途停止后旧目标造成方向状态残留。
//
// 调用位置：
// 必须在M_UpdateMotionState和M_UpdateAxisData之后调用。
//==============================================================

METHOD PRIVATE M_UpdateMotionDirection

VAR_IN_OUT
    ioAxis : ST_AxisInterface;
    // 当前单轴命令、数据和状态接口
END_VAR

VAR CONSTANT
    // 速度方向判断死区。
    //
    // 防止轴在零速附近因浮点波动频繁切换正负方向。
    // 当前单位取决于具体业务轴的工程单位，直线轴通常为mm/s。
    c_fVelocityDeadband : LREAL := GVL_MotionConfig.fAxisDirectionVelocityDeadband;
END_VAR

VAR
    // 最终用于判断正负方向的速度。
    fDirectionVelocity : LREAL;
END_VAR
//==============================================================
// 1. 每周期默认清除方向
//
// 先写None可以保证：
// 1. 轴停止后不会保留上一次运动方向；
// 2. 故障、掉使能和复位时不会显示旧方向；
// 3. 方法后续即使没有满足方向条件，状态也始终明确。
//==============================================================

ioAxis.State.eMotionDirection :=
    E_AxisMotionDirection.None;


//==============================================================
// 2. 只在定位运动或点动期间判断方向
//
// Stopping状态由WPF显示为“停止中”；
// Standstill状态由WPF显示为“停止”；
// 因此这些状态不再输出Positive或Negative。
//==============================================================

IF
    (ioAxis.State.eMotionState = E_AxisMotionState.Moving)
    OR
    (ioAxis.State.eMotionState = E_AxisMotionState.Homing)
    OR
    (ioAxis.State.eMotionState = E_AxisMotionState.Jogging)
    OR
    (ioAxis.State.eMotionState = E_AxisMotionState.TorqueRunning)
THEN

    //==========================================================
    // 3. 优先使用实际速度
    //
    // 实际速度能够反映轴真正运动的方向，
    // 不会受到旧目标位置或点动NC目标位置的影响。
    //==========================================================

    fDirectionVelocity :=
        ioAxis.Data.fActVelocity;


    //==========================================================
    // 4. 实际速度尚未建立时使用设定速度
    //
    // 运动命令刚被接受的前几个PLC周期中，
    // eMotionState可能已经是Moving或Jogging，
    // 但实际速度仍然接近0。
    //
    // 此时使用NC设定速度可以尽早显示运动方向。
    //==========================================================

    IF
        ABS(fDirectionVelocity)
        <= c_fVelocityDeadband
    THEN

        fDirectionVelocity :=
            ioAxis.Data.fSetVelocity;

    END_IF;


    //==========================================================
    // 5. 根据速度正负生成统一方向状态
    //==========================================================

    IF
        fDirectionVelocity
        > c_fVelocityDeadband
    THEN

        ioAxis.State.eMotionDirection :=
            E_AxisMotionDirection.Positive;

    ELSIF
        fDirectionVelocity
        < -c_fVelocityDeadband
    THEN

        ioAxis.State.eMotionDirection :=
            E_AxisMotionDirection.Negative;

    ELSE

        // Moving/Jogging已经建立，但实际速度和设定速度
        // 暂时都处于零速死区，例如刚启动或即将停止。
        ioAxis.State.eMotionDirection :=
            E_AxisMotionDirection.None;

    END_IF;

END_IF;
END_METHOD

//==============================================================
// 方法名称：M_UpdateMotionState
// 功能：根据轴错误、停止、复位、点动、定位和使能状态，
//       生成唯一的E_AxisMotionState运动状态。
//
// 状态优先级：
// Error > Stopping > Resetting > Jogging > Moving
// > Disabled > NotReady > Standstill
//
// 调用位置：
// 必须放在执行方法、错误汇总和基础状态更新之后。
//==============================================================

METHOD PRIVATE M_UpdateMotionState

VAR_IN_OUT
    ioAxisRef : AXIS_REF;
    // 当前TwinCAT NC轴引用

    ioAxis : ST_AxisInterface;
    // 当前单轴状态和报警接口
END_VAR
//==============================================================
// 1. 错误状态
//
// NC轴错误或PLC锁存错误存在时，统一进入Error。
//==============================================================

IF
    ioAxisRef.Status.Error
    OR ioAxis.Alarm.bError
THEN

    ioAxis.State.eMotionState :=
        E_AxisMotionState.Error;


//==============================================================
// 2. 停止状态
//
// stInternal.bStopExecute包含Stop已经锁存但Busy尚未建立的阶段。
//==============================================================

ELSIF
    stInternal.bStopExecute
    OR fbStop.Busy
THEN

    ioAxis.State.eMotionState :=
        E_AxisMotionState.Stopping;


//==============================================================
// 3. 复位状态
//==============================================================

ELSIF fbReset.Busy THEN

    ioAxis.State.eMotionState :=
        E_AxisMotionState.Resetting;


//==============================================================
// 4. 回零状态
//==============================================================

ELSIF
    fbHome.Busy
    OR stInternal.bHomeExecute
THEN

    ioAxis.State.eMotionState :=
        E_AxisMotionState.Homing;


//==============================================================
// 5. 转矩控制状态
//==============================================================

ELSIF
    fbTorqueControl.Active
    OR fbTorqueControl.Busy
    OR stInternal.bTorqueExecute
THEN

    ioAxis.State.eMotionState :=
        E_AxisMotionState.TorqueRunning;


//==============================================================
// 5. 点动状态
//==============================================================

ELSIF fbJog.Busy THEN

    ioAxis.State.eMotionState :=
        E_AxisMotionState.Jogging;


//==============================================================
// 6. 定位运动状态
//
// Execute锁存可以覆盖命令已接受但Busy尚未建立的周期。
//==============================================================

ELSIF
    fbMoveAbs.Busy
    OR fbMoveRel.Busy
    OR stInternal.bMoveAbsExecute
    OR stInternal.bMoveRelExecute
THEN

    ioAxis.State.eMotionState :=
        E_AxisMotionState.Moving;


//==============================================================
// 7. 未使能状态
//==============================================================

ELSIF NOT fbPower.Status THEN

    ioAxis.State.eMotionState :=
        E_AxisMotionState.Disabled;


//==============================================================
// 8. 控制未许可状态
//
// 轴已经使能，但外部控制许可无效。
//==============================================================

ELSIF NOT bControlAllowed THEN

    ioAxis.State.eMotionState :=
        E_AxisMotionState.NotReady;


//==============================================================
// 9. 静止状态
//
// 轴已使能、控制许可有效、无错误且没有执行命令。
//==============================================================

ELSE

    ioAxis.State.eMotionState :=
        E_AxisMotionState.Standstill;

END_IF;
END_METHOD

//==============================================================
// 方法名称：M_UpdateSoftLimitState
//
// 功能：
// 1. 检查软件限位配置是否合法；
// 2. 检查当前坐标基准是否有效；
// 3. 计算正负点动方向许可；
// 4. 检查绝对运动目标；
// 5. 计算并检查相对运动最终目标；
// 6. 更新WPF所需的软件限位状态。
//
// 注意：
// 1. 本方法只计算状态，不调用任何MC功能块；
// 2. 相对运动必须基于NC设定位置SetPos计算；
// 3. 已经超限时，禁止继续向外，但允许向内返回。
//==============================================================

METHOD PRIVATE M_UpdateSoftLimitState

VAR_INPUT
    iLimit : ST_AxisLimit;
    // 当前轴的软件限位配置
END_VAR

VAR_IN_OUT
    ioAxisRef : AXIS_REF;
    // 当前NC轴引用

    ioAxis : ST_AxisInterface;
    // 当前单轴接口
END_VAR
//==============================================================
// 1. 读取是否启用软件限位
//==============================================================

stInternal.stSoftLimitResult.bEnabled :=
    iLimit.bSoftLimitEnable;


//==============================================================
// 2. 检查限位配置
//
// 配置必须满足：
// 1. 负限位小于正限位；
// 2. Margin不能为负数；
// 3. 两侧Margin之间仍然存在有效运动范围。
//==============================================================

stInternal.stSoftLimitResult.bConfigValid :=
    iLimit.fSoftwareLimitNeg
        < iLimit.fSoftwareLimitPos

    AND iLimit.fSoftLimitMargin >= 0.0

    AND
    (
        iLimit.fSoftwareLimitNeg
        + iLimit.fSoftLimitMargin
    )
    <
    (
        iLimit.fSoftwareLimitPos
        - iLimit.fSoftLimitMargin
    );


//==============================================================
// 3. 检查坐标基准
//
// 不要求回零时，坐标基准直接视为有效。
// 要求回零时，必须等待AxisRef.Status.Homed为TRUE。
//==============================================================

stInternal.stSoftLimitResult.bReferenceValid :=
    NOT iLimit.bRequireHomed
    OR ioAxisRef.Status.Homed;


//==============================================================
// 4. 汇总软件限位是否可用
//
// 禁用软限位时，不阻止任何运动。
// 启用时，配置和坐标基准必须同时有效。
//==============================================================

stInternal.stSoftLimitResult.bReady :=
    NOT stInternal.stSoftLimitResult.bEnabled
    OR
    (
        stInternal.stSoftLimitResult.bConfigValid
        AND stInternal.stSoftLimitResult.bReferenceValid
    );


//==============================================================
// 5. 计算相对运动最终目标
//
// MC_MoveRelative以当前NC设定位置SetPos为基准。
// 不应使用ActPos计算相对运动最终目标。
//==============================================================

stInternal.stSoftLimitResult.fRelativeTargetPosition :=
    ioAxisRef.NcToPlc.SetPos
    + ioAxis.ActiveSet.Position.fRelativeDistance;


//==============================================================
// 6. 软件限位未启用
//
// 所有运动方向和目标均允许。
//==============================================================

IF NOT stInternal.stSoftLimitResult.bEnabled THEN

    stInternal.stSoftLimitResult.bPositiveActive := FALSE;
    stInternal.stSoftLimitResult.bNegativeActive := FALSE;

    stInternal.stSoftLimitResult.bJogPositiveAllowed := TRUE;
    stInternal.stSoftLimitResult.bJogNegativeAllowed := TRUE;

    stInternal.stSoftLimitResult.bAbsoluteTargetValid := TRUE;
    stInternal.stSoftLimitResult.bRelativeTargetValid := TRUE;


//==============================================================
// 7. 软件限位启用且状态有效
//==============================================================

ELSIF stInternal.stSoftLimitResult.bReady THEN

    // 使用实际位置生成WPF限位指示
    stInternal.stSoftLimitResult.bPositiveActive :=
        ioAxisRef.NcToPlc.ActPos
        >=
        (
            iLimit.fSoftwareLimitPos
            - iLimit.fSoftLimitMargin
        );

    stInternal.stSoftLimitResult.bNegativeActive :=
        ioAxisRef.NcToPlc.ActPos
        <=
        (
            iLimit.fSoftwareLimitNeg
            + iLimit.fSoftLimitMargin
        );


    // 正向点动进入正向缓冲区域后停止继续向外运动
    stInternal.stSoftLimitResult.bJogPositiveAllowed :=
        ioAxisRef.NcToPlc.SetPos
        <
        (
            iLimit.fSoftwareLimitPos
            - iLimit.fSoftLimitMargin
        );


    // 负向点动进入负向缓冲区域后停止继续向外运动
    stInternal.stSoftLimitResult.bJogNegativeAllowed :=
        ioAxisRef.NcToPlc.SetPos
        >
        (
            iLimit.fSoftwareLimitNeg
            + iLimit.fSoftLimitMargin
        );


    // 检查绝对目标
    stInternal.stSoftLimitResult.bAbsoluteTargetValid :=
        ioAxis.ActiveSet.Position.fAbsolutePosition
            >= iLimit.fSoftwareLimitNeg
        AND
        ioAxis.ActiveSet.Position.fAbsolutePosition
            <= iLimit.fSoftwareLimitPos;


    // 检查相对运动计算得到的最终目标
    stInternal.stSoftLimitResult.bRelativeTargetValid :=
        stInternal.stSoftLimitResult.fRelativeTargetPosition
            >= iLimit.fSoftwareLimitNeg
        AND
        stInternal.stSoftLimitResult.fRelativeTargetPosition
            <= iLimit.fSoftwareLimitPos;


//==============================================================
// 8. 软件限位启用但配置或坐标基准无效
//
// 采用失效安全原则，禁止普通运动。
//==============================================================

ELSE

    stInternal.stSoftLimitResult.bPositiveActive := FALSE;
    stInternal.stSoftLimitResult.bNegativeActive := FALSE;

    stInternal.stSoftLimitResult.bJogPositiveAllowed := FALSE;
    stInternal.stSoftLimitResult.bJogNegativeAllowed := FALSE;

    stInternal.stSoftLimitResult.bAbsoluteTargetValid := FALSE;
    stInternal.stSoftLimitResult.bRelativeTargetValid := FALSE;

END_IF;


//==============================================================
// 9. 更新WPF状态反馈
//==============================================================

ioAxis.State.bSoftLimitEnabled :=
    stInternal.stSoftLimitResult.bEnabled;

ioAxis.State.bSoftLimitReady :=
    stInternal.stSoftLimitResult.bReady;

ioAxis.State.bSoftLimitPositive :=
    stInternal.stSoftLimitResult.bPositiveActive;

ioAxis.State.bSoftLimitNegative :=
    stInternal.stSoftLimitResult.bNegativeActive;
END_METHOD

END_FUNCTION_BLOCK

(* stored: Version 1.1.0.1, ProductVersion 3.1.4026.18
   POU FB_AxisControl: Id {cbe667f4-3a4a-4731-acdb-ae88eb96b09a}, SpecialFunc None
   Method M_ClearCycleResults: Id {b0100f26-6f1e-463a-8206-ad01d5a00796}
   Method M_ExecuteHoming: Id {71335fbe-04e0-4534-b1dc-a74e79e4fd26}
   Method M_ExecuteJog: Id {a4ee27c3-dd78-49f1-a96d-8089113d52a3}
   Method M_ExecutePositioning: Id {f6694070-471f-441e-a9e8-b34f3a930dbc}
   Method M_ExecuteTorqueControl: Id {8f59c356-6219-4eab-b050-e71d0c124f35}
   Method M_ExecutePowerReset: Id {97d51e5c-08e7-4f36-a4c4-b68d43d17128}
   Method M_ExecuteStop: Id {b3e2f5b9-520d-444d-9b18-5c763a9aea1b}
   Method M_ReadAxisStatus: Id {d0e5ee8d-228a-4964-9d8c-da9887885914}
   Method M_SelectCommand: Id {3eba9e33-1af3-4d6b-bf6d-4e9299aa666b}
   Method M_UpdateAxisData: Id {90593075-838c-4824-af74-478ff719ba9d}
   Method M_UpdateBasicState: Id {5450b6ce-a3d6-4d3c-84ee-f95ee610611d}
   Method M_UpdateCommandArbitration: Id {d8b16562-dea7-412c-a822-b092e5d2cca8}
   Method M_UpdateCommandEdges: Id {4c7b1159-4005-4e07-bab0-2bc66c855e7f}
   Method M_UpdateError: Id {dd0c9f2b-f27c-4abb-b438-65065b8f3756}
   Method M_UpdateMotionDirection: Id {ef82fa8e-8387-4d59-b60a-cdad9b7d7a20}
   Method M_UpdateMotionState: Id {f24094b2-eed5-45d6-807b-d5bb6e886654}
   Method M_UpdateSoftLimitState: Id {072cd1fa-f091-44c5-8764-82398ddee6ea} *)
